// TIA Portal V18 export
TYPE "PosList"
// stored: IsFailsafeCompliant false
   STRUCT
      List : Array[0..39] of Struct
         Pos : DInt;
         Vel : Int;
      END_STRUCT;
   END_STRUCT;
END_TYPE
